# B&R Automation Studio project Projekt_BuR
Automation Studio 4.11.2.75; technology packages: exosTechnology 2.1.0, mapp 5.18.0, mappCockpit 5.18.0, mappControl 5.18.0, mappView 5.18.1

## Configuration X20CP3586

CPU X20CP3586, AutomationRuntime C4.92, Build 4.1.2, Safety 0.0, Vc V4.72.5

### Task classes (Cpu.sw)
```
Cyclic#1 (cycle 2000 us, tolerance 0 us):
  TempContro <- Control.TempControl.prg
  TempScalin <- TempScaling.prg
Cyclic#3:
  MQTT <- Control.MQTT.prg
Cyclic#4:
  Alarm <- Control.Alarm.prg
  Recipe <- Control.Recipe.prg
  OEE <- Control.OEE.prg
  AuditTrail <- Control.AuditTrail.prg
  MpReport1 <- Control.MpReport.prg
  DataMgmt <- Control.DataMgmt.prg
  VisuAdj <- Control.VisuAdj.prg
  FileCtrl <- Control.FileCtrl.prg
Binaries: udbdef, FWRules, TCData, TCLang, arsvcreg, mvLoader, mCoWebSc, arflatprv, arcoal, iomap, ashwac, Role, sysconf, arconfig, asfw, User, ashwd, HeatZone3, HeatZone2, HeatZone1, HeatZone4, TC, HeatGroup, ConfigAudi, ConfigAHis, ConfigAlar, ConfigData, ConfigOEE, report, ConfigFile, RecipeCon, Config
Libraries: CoTrace, AsZip, FileIO, runtime, MpAlarmX, MpBase, astime, MpServer, MpTemp, IotMqtt, AsIecCon, ArCert, sys_lib, AsHW, AsETH, ArEventLog, AsIODiag, AsBrStr, standard, MpAudit, MpReport, AsMath, MpOee, MpData, DataObj, brsystem, MpFile, MpRecipe, MTBasics, MTTypes, arssl, aruser, asusb, MpUserX
```

### Hardware
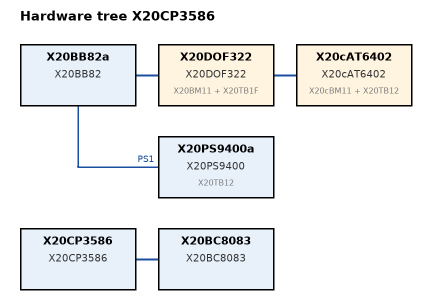
```
X20BB82a : X20BB82 v1.1.0.0
X20BC8083 : X20BC8083 v2.12.0.0  [PLK1 -> X20CP3586.IF3 (NodeNumber=1) [Cable Type=PowerlinkCable, Length=10, Version=1.0.0.3]; SL -> X20BB82a.SL1]
  Supervision = off
X20BM11a : X20BM11 v1.1.0.0  [X2X1 -> X20BB82a.IF1]
X20CP3586 : X20CP3586 v1.10.0.0
  Connector IF2:
    ActivateDevice = 1
    Mode = Manual
    InternetAddress = 192.168.0.22
    SubnetMask = 255.255.255.0
    ActivateSnmp = 2
  Connector IF3:
    CycleTime = 400
  ConfigurationID = Projekt_BuR_X20CP3586
  TimerDeviceType = EPLX2X
  TimerDevice = X20CP3586.IF3
  TaskClassIdleTime = 2000
  Cyclic1Duration = 2000
  Cyclic1Tolerance = 0
  FileDevice1
  FileDeviceName1 = AUDIT
  FileDevicePath1 = F:/BRAudit
  FileDevice2
  FileDeviceName2 = DATA
  FileDevicePath2 = F:/BRmappData
  FileDevice3
  FileDeviceName3 = PDF
  FileDevicePath3 = F:/PDF
  FileDevice4
  FileDeviceName4 = DISK
  FileDevicePath4 = F:/
  FileDevice5
  FileDeviceName5 = RECIPE
  FileDevicePath5 = F:/BrRecipe
  FileDevice6
  FileDeviceName6 = BRVisu
  FileDevicePath6 = C:/ADDONS/DATA/IAT_Data/wwwRoot/BRVisu
  TimeZone = 160
  ActivateDaylightSavingTime = 1
  FtpUser1
  FtpUsername1 = Admin
  FtpUserPassword1 = 5wGvT8auoKyFZyijp5IHEBz1PpSmCNNWGV/kzWv0+cU=
  FtpUserSalt1 = OGipJzaF
  FTPAccessRight1 = 0
  FTPdevice1 = ALL
  ActivateOpcUa = 1
  OpcUaInformationModels_PV_Version = 1
X20DOF322 : X20DOF322 v1.5.0.0  [SS1 -> X20TB1F1.SS; SL -> X20BM11a.SL1]
  Supervision = off
X20PS9400a : X20PS9400 v1.7.0.0  [SS1 -> X20TB12.SS; PS -> X20BB82a.PS1]
  Supervision = off
X20TB12 : X20TB12 v1.0.0.0
X20TB12a : X20TB12 v1.0.0.0
X20TB1F1 : X20TB1F v1.0.0.0
X20cAT6402 : X20cAT6402 v1.2.0.0  [SS1 -> X20TB12a.SS; SL -> X20cBM11a.SL1]
  Supervision = off
  DisableChannel01 = on
  DisableChannel02 = on
X20cBM11a : X20cBM11 v1.1.0.0  [X2X1 -> X20BM11a.X2X2]
```

### ConfigAlar.mpalarmxcore - X20CP3586/mappServices/ConfigAlar.mpalarmxcore
```
Element gAlarmXCore (Type=mpalarmxcore)
  mapp.AlarmX.Core:
    Mapping:
      [0]:
        Alarm = High Temperature1#HighHigh
        [0] = Reaction
          Name = StatusIdle
      [1]:
        Alarm = High Temperature2#HighHigh
        [0] = Reaction
          Name = StatusIdle
      [2]:
        Alarm = High Temperature3#HighHigh
        [0] = Reaction
          Name = StatusIdle
      [3]:
        Alarm = High Temperature4#HighHigh
        [0] = Reaction
          Name = StatusIdle
      [4]:
        Alarm = X20BC8083
        [0] = Reaction
          Name = StatusIdle
      [5]:
        Alarm = X20PS9400a
        [0] = Reaction
          Name = StatusIdle
      [6]:
        Alarm = X20DOF322
        [0] = Reaction
          Name = StatusIdle
      [7]:
        Alarm = X20cAT6402
        [0] = Reaction
          Name = StatusIdle
      [8]:
        Alarm =  Fan failure1
        [0] = Reaction
          Name = StatusIdle
      [9]:
        Alarm =  Fan failure2
        [0] = Reaction
          Name = StatusIdle
      [10]:
        Alarm =  Fan failure3
        [0] = Reaction
          Name = StatusIdle
      [11]:
        Alarm =  Fan failure4
        [0] = Reaction
          Name = StatusIdle
      [12]:
        Alarm = Sensor failure1
        [0] = Reaction
          Name = StatusIdle
      [13]:
        Alarm = Sensor failure2
        [0] = Reaction
          Name = StatusIdle
      [14]:
        Alarm = Sensor failure3
        [0] = Reaction
          Name = StatusIdle
      [15]:
        Alarm = Sensor failure4
        [0] = Reaction
          Name = StatusIdle
  mapp.AlarmX.Core.Configuration:
    [0]:
      Name = High Temperature1
      Message = {$IAT/Alarms/HT1Message}
      Code = 1037
      Behavior = LevelMonitoring
        Monitoring:
          MonitoredPV = ::gTemp1
          HighLimitEnable = Dynamic
            LimitPV = ::Alarms.TempAlarmLimit
            HighHighLimitEnable = Dynamic
              LimitPV = ::Alarms.TempMaxAlarmLimit
              LimitText = HighHigh
    [1]:
      Name = High Temperature2
      Message = {$IAT/Alarms/HT2Message}
      Code = 1038
      Behavior = LevelMonitoring
        Monitoring:
          MonitoredPV = ::gTemp2
          HighLimitEnable = Dynamic
            LimitPV = ::Alarms.TempAlarmLimit
            HighHighLimitEnable = Dynamic
              LimitPV = ::Alarms.TempMaxAlarmLimit
              LimitText = HighHigh
    [2]:
      Name = High Temperature3
      Message = {$IAT/Alarms/HT3Message}
      Code = 1039
      Behavior = LevelMonitoring
        Monitoring:
          MonitoredPV = ::gTemp3
          HighLimitEnable = Dynamic
            LimitPV = ::Alarms.TempAlarmLimit
            HighHighLimitEnable = Dynamic
              LimitPV = ::Alarms.TempMaxAlarmLimit
              LimitText = HighHigh
    [3]:
      Name = High Temperature4
      Message = {$IAT/Alarms/HT4Message}
      Code = 1040
      Behavior = LevelMonitoring
        Monitoring:
          MonitoredPV = ::gTemp4
          HighLimitEnable = Dynamic
            LimitPV = ::Alarms.TempAlarmLimit
            HighHighLimitEnable = Dynamic
              LimitPV = ::Alarms.TempMaxAlarmLimit
              LimitText = HighHigh
    [4]:
      Name = X20BC8083
      Message = {$IAT/Alarms/X20BC8083}
      Code = 1308
      Behavior = DiscreteValueMonitoring
        Monitoring:
          MonitoredPV = ::Alarms.first_module
          TriggerValues:
            [0] = 0
    [5]:
      Name = X20PS9400a
      Message = {$IAT/Alarms/X20PS9400a}
      Code = 1309
      Behavior = DiscreteValueMonitoring
        Monitoring:
          MonitoredPV = ::Alarms.second_module
          TriggerValues:
            [0] = 0
    [6]:
      Name = X20DOF322
      Message = {$IAT/Alarms/X20DOF322}
      Code = 1310
      Behavior = DiscreteValueMonitoring
        Monitoring:
          MonitoredPV = ::Alarms.third_module
          TriggerValues:
            [0] = 0
    [7]:
      Name = X20cAT6402
      Message = {$IAT/Alarms/X20cAT6402}
      Code = 1311
      Behavior = DiscreteValueMonitoring
        Monitoring:
          MonitoredPV = ::Alarms.fourth_module
          TriggerValues:
            [0] = 0
    [8]:
      Name =  Fan failure1
      Message = {$IAT/Alarms/FanAlarmMessage1}
      Code = 1446
      Behavior = DiscreteValueMonitoring
        Monitoring:
          MonitoredPV = ::Alarms.FanAlarm1
          TriggerValues:
            [0] = 1
    [9]:
      Name =  Fan failure2
      Message = {$IAT/Alarms/FanAlarmMessage2}
      Code = 1447
      Behavior = DiscreteValueMonitoring
        Monitoring:
          MonitoredPV = ::Alarms.FanAlarm2
          TriggerValues:
            [0] = 1
    [10]:
      Name =  Fan failure3
      Message = {$IAT/Alarms/FanAlarmMessage3}
      Code = 1448
      Behavior = DiscreteValueMonitoring
        Monitoring:
          MonitoredPV = ::Alarms.FanAlarm3
          TriggerValues:
            [0] = 1
    [11]:
      Name =  Fan failure4
      Message = {$IAT/Alarms/FanAlarmMessage4}
      Code = 1449
      Behavior = DiscreteValueMonitoring
        Monitoring:
          MonitoredPV = ::Alarms.FanAlarm4
          TriggerValues:
            [0] = 1
    [12]:
      Name = Sensor failure1
      Message = {$IAT/Alarms/HeaterAlarmMess1}
      Severity = 1455
      Behavior = DiscreteValueMonitoring
        Monitoring:
          MonitoredPV = ::Alarms.HeaterAlarm1
          TriggerValues:
            [0] = 1
    [13]:
      Name = Sensor failure2
      Message = {$IAT/Alarms/HeaterAlarmMess2}
      Severity = 1456
      Behavior = DiscreteValueMonitoring
        Monitoring:
          MonitoredPV = ::Alarms.HeaterAlarm2
          TriggerValues:
            [0] = 1
    [14]:
      Name = Sensor failure3
      Message = {$IAT/Alarms/HeaterAlarmMess3}
      Severity = 1457
      Behavior = DiscreteValueMonitoring
        Monitoring:
          MonitoredPV = ::Alarms.HeaterAlarm3
          TriggerValues:
            [0] = 1
    [15]:
      Name = Sensor failure4
      Message = {$IAT/Alarms/HeaterAlarmMess4}
      Severity = 1458
      Behavior = DiscreteValueMonitoring
        Monitoring:
          MonitoredPV = ::Alarms.HeaterAlarm4
          TriggerValues:
            [0] = 1
```

### ConfigUser.mpuserx - X20CP3586/mappServices/ConfigUser.mpuserx
```
Element UserMgmtX (Type=mpuserx)
  ServerSettings:
    Server:
      AdditionalUserData:
        [0] = mail
        [1] = telephoneNumber
  Users:
    DefUser#1:
      id = Administrator
    DefUser#2:
      id = Operator
    DefUser#3:
      id = a
    DefUser#4:
      id = Anonymous
  Groups:
    DefGroup#1:
      id = Administrators
      level = 100
      admin = TRUE
      rights:
        [0] = FullAccess
    DefGroup#2:
      id = Operators
      level = 30
    DefGroup#3:
      id = Everyone
      level = 3
```

## Logical view

Binary libraries used (declarations not repeated): operator, runtime, astime, AsIecCon, CoTrace, AsZip, FileIO, MpAlarmX, MpBase, MpServer, MpTemp, IotMqtt, ArCert, sys_lib, AsHW, AsETH, ArEventLog, AsIODiag, AsBrStr, standard, MpOee, MpAudit, MpReport, AsMath, MpData, DataObj, brsystem, MpFile, MpRecipe, MTBasics, MTTypes, MpUserX, ExOS, ExDeploy, ExData, AsIoTime

### ControlTypes.typ
```iecst
TYPE
	AUTOMATIC_MODE_STATE :
		( (*Step of automatic mode*)
		STEP_INIT,
		STEP1,
		STEP2,
		STEP3,
		STEP4,
		STEP5
		);
	ZONE_WORKING_STATE :
		( (*Working state of each zone*)
		STATE_IDLE_ZONE,
		STATE_HEATING,
		STATE_COOLING
		);
	MACHINE_WORKING_STATE :
		( (*Working state of whole machine*)
		STATE_IDLE,
		STATE_TUNING,
		STATE_WORKING_MANUAL,
		STATE_WORKING_AUTOMATIC,
		STATE_ERROR,
		STATE_STOP
		);
	MACHINE_PARAMETERS : 	STRUCT  (*Machine parameters - structed*)
		Temp1 : REAL;
		Temp2 : REAL;
		Temp3 : REAL;
		Temp4 : REAL;
		Time1 : TIME;
		Time2 : TIME;
		Time3 : TIME;
		Time4 : TIME;
		Time5 : TIME;
	END_STRUCT;
	Alarm_struct : 	STRUCT
		Pending : UDINT := 0;
		Active : UDINT := 0;
		FanAlarm4 : BOOL;
		FanAlarm3 : BOOL;
		FanAlarm2 : BOOL;
		FanAlarm1 : BOOL;
		HeaterAlarm4 : BOOL;
		HeaterAlarm3 : BOOL;
		HeaterAlarm2 : BOOL;
		HeaterAlarm1 : BOOL;
		fourth_module : BOOL;
		third_module : BOOL;
		second_module : BOOL;
		first_module : BOOL;
		TempMaxAlarmLimit : REAL := 50;
		TempAlarmLimit : REAL := 40;
		ActiveAlarms : STRING[512] := 'test';
	END_STRUCT;
	OEE_Struct : 	STRUCT
		IdealCycleTime : STRING[80];
		OEE : REAL;
		Quality : REAL;
		Performance : REAL;
		Availability : REAL;
		RejectCounter : UDINT;
		PieceCounter : UDINT;
	END_STRUCT;
END_TYPE
```

### ControlVariables.var
```iecst
(*Temperature setpoints to all zones.*)
VAR
	SetTemp1 : REAL := 30; (*Set temperature for zone 1.*)
	SetTemp2 : REAL := 30; (*Set temperature for zone 2.*)
	SetTemp3 : REAL := 30; (*Set temperature for zone 3.*)
	SetTemp4 : REAL := 30; (*Set temperature for zone 4.*)
END_VAR
(*Temperature tuning setpoints to all zones.*)
VAR
	SetTempHeatTuning1 : REAL := 100; (*Set heating temperature for zone 1.*)
	SetTempHeatTuning2 : REAL := 100; (*Set heating temperature for zone 2.*)
	SetTempHeatTuning3 : REAL := 100; (*Set heating temperature for zone 3.*)
	SetTempHeatTuning4 : REAL := 100; (*Set  heating temperature for zone 4.*)
	SetTempCoolTuning1 : REAL := 30; (*Set cooling temperature for zone 1.*)
	SetTempCoolTuning2 : REAL := 30; (*Set cooling temperature for zone 2.*)
	SetTempCoolTuning3 : REAL := 30; (*Set cooling temperature for zone 3.*)
	SetTempCoolTuning4 : REAL := 30; (*Set cooling temperature for zone 4.*)
END_VAR
(*Machine status - step.*)
VAR
	STATUS : MACHINE_WORKING_STATE := STATE_IDLE; (*Whole machine working status.*)
END_VAR
(*Zones status*)
VAR
	ZoneStatus : ARRAY[0..ELEMENTS_NUMBER] OF ZONE_WORKING_STATE; (*Each zone working status.*)
END_VAR
(*Temperature controller functionblocks.*)
VAR
	TempControllerPar : ARRAY[0..ELEMENTS_NUMBER] OF MpTempControllerParType; (*Array of 4 additions to controllers*)
	TempController : ARRAY[0..ELEMENTS_NUMBER] OF MpTempController; (*Array of 4 controllers - one for each zone*)
	TempGroup : MpTempGroup; (*Controller group*)
	TempGroupPar : MpTempGroupParType; (*Adition to controllergroup*)
END_VAR
(*Const elements.*)
VAR CONSTANT
	ELEMENTS_NUMBER : USINT := 3; (*Numbers of controling zones - 4 (0,1,2,3)*)
END_VAR
(*Machine working type*)
VAR
	Automatic_work : BOOL := FALSE; (*Enable automatic work mode.*)
	Manual_work : BOOL := FALSE; (*Enable manual work mode.*)
	TuneEnable : BOOL := FALSE; (*Enable tune work mode.*)
END_VAR
(*Manual control*)
VAR
	EnableZone1 : BOOL := TRUE; (*Enable zone 1.*)
	EnableZone2 : BOOL := TRUE; (*Enable zone 2.*)
	EnableZone3 : BOOL := TRUE; (*EnableZone 3.*)
	EnableZone4 : BOOL := TRUE; (*Enable zone 4.*)
END_VAR
(*Automatic control*)
VAR
	AutoStep : AUTOMATIC_MODE_STATE := STEP_INIT;
	TimeStep1 : TIME := T#5s; (*Min time of step 1*)
	TimeStep2 : TIME := T#5s; (*Min time of step 2*)
	TimeStep3 : TIME := T#5s; (*Min time of step 3*)
	TimeStep4 : TIME := T#5s; (*Min time of step 4*)
	TimeStep5 : TIME := T#5s; (*Min time of step 5*)
	TimStep1 : TON; (*Timer for step 1 in automatic work.*)
	TimStep2 : TON; (*Timer for step 2 in automatic work.*)
	TimStep3 : TON; (*Timer for step 3 in automatic work.*)
	TimStep4 : TON; (*Timer for step 4 in automatic work.*)
	TimStep5 : TON; (*Timer in step 5 for automatic work.*)
	CycleNumber : DINT := 0; (*Number of full done cycles in automatic work.*)
END_VAR
(*Simulation mode*)
VAR
	SimulateZone1Enable : BOOL := FALSE; (*Simulation enable of zone 1.*)
	SimulateZone2Enable : BOOL := FALSE; (*Simulation enable of zone 2.*)
	SimulateZone3Enable : BOOL := FALSE; (*Simulation enable of zone 3.*)
	SimulateZone4Enable : BOOL := FALSE; (*Simulation enable of zone 4.*)
END_VAR
(*Tuning parameters HEAT*)
VAR RETAIN
	PIDProportionaGainHEAT : ARRAY[0..ELEMENTS_NUMBER] OF REAL := [49.3,45.56,31.29,35.25];
	PIDIntegrationTimeHEAT : ARRAY[0..ELEMENTS_NUMBER] OF REAL := [64.92,75.59,95.21,101.41];
	PIDFilterTimeHEAT : ARRAY[0..ELEMENTS_NUMBER] OF REAL := [0.682,0.762,0.99,1.06];
	PIDDerivativeTimeHEAT : ARRAY[0..ELEMENTS_NUMBER] OF REAL := [6.82,7.62,9.99,10.64];
END_VAR
(*Tuning parameters COOL*)
VAR RETAIN
	PIDProportionaGainCOOL : ARRAY[0..ELEMENTS_NUMBER] OF REAL := [20.96,27.64,18.07,26.18];
	PIDIntegrationTimeCOOL : ARRAY[0..ELEMENTS_NUMBER] OF REAL := [68.71,46.86,80.30,51.64];
	PIDDerivativeTimeCOOL : ARRAY[0..ELEMENTS_NUMBER] OF REAL := [7.22,4.92,8.43,5.42];
	PIDFilterTimeCOOL : ARRAY[0..ELEMENTS_NUMBER] OF REAL := [0.72,0.49,0.84,0.54];
END_VAR
(*Alarm*)
VAR
	Alarms : Alarm_struct;
	MpAlarmXCore_0 : MpAlarmXCore;
END_VAR
(*OEE*)
VAR
	OEE : OEE_Struct;
END_VAR
(* ########## MQTT communication variables ########### *)
(*PWM % Heater Zone 1  ->  TempController[0].HeatValue*)
(*PWM % Heater Zone 2  ->  TempController[1].HeatValue*)
(*PWM % Heater Zone 3  ->  TempController[2].HeatValue*)
(*PWM % Heater Zone 4  ->  TempController[3].HeatValue*)
(*PWM % FAN Zone 1  ->  TempController[0].CoolValue*)
(*PWM % FAN Zone 2  ->  TempController[1].CoolValue*)
(*PWM % FAN Zone 3  ->  TempController[2].CoolValue*)
(*PWM % FAN Zone 4  ->  TempController[3].CoolValue*)
(*Set Temperature Zone 1  ->  SetTemp1*)
(*Set Temperature Zone 2  ->  SetTemp2*)
(*Set Temperature Zone 3  ->  SetTemp3*)
(*Set Temperature Zone 4  ->  SetTemp4*)
(*Actual Temperature Zone 1  ->  gTemp1*)
(*Actual Temperature Zone 2  ->  gTemp2*)
(*Actual Temperature Zone 3  ->  gTemp3*)
(*Actual Temperature Zone 4  ->  gTemp4*)
(*Status dzialania calej maszyny -> STATUS (typ: MACHINE_WORKING_STATE)*)
(*Status dzialania trybu automatycznego -> AutoStep (typ: AUTOMATIC_MODE_STATUS)*)
(*Status dzialania strefy 1 -> ZoneStatus[0] (typ: ZONE_WORKING_STATUS)*)
(*Status dzialania strefy 2 -> ZoneStatus[1] (typ: ZONE_WORKING_STATUS)*)
(*Status dzialania strefy 3 -> ZoneStatus[2] (typ: ZONE_WORKING_STATUS)*)
(*Status dzialania strefy 4 -> ZoneStatus[3] (typ: ZONE_WORKING_STATUS)*)
(*Ilosc wykonanych cykli w trybie automatycznym -> CycleNumber*)
(*//////////////////////////////Machine parameters*)
VAR
	ParametersMachine : MACHINE_PARAMETERS;
END_VAR
(*Recipe*)
VAR
	RecipeListName : ARRAY[0..9] OF STRING[255];
END_VAR
(*Audit*)
VAR
	MpAuditTrail_0 : MpAuditTrail;
	MessageVar : WSTRING[100] := "Hello World";
END_VAR
(*pid pwm*)
VAR
	MTBasicsPID_HEAT : ARRAY[0..ELEMENTS_NUMBER] OF MTBasicsPID;
	ParameterTypePIDHEAT : ARRAY[0..ELEMENTS_NUMBER] OF MTPIDParametersType;
	MTBasicsPID_COLD : ARRAY[0..ELEMENTS_NUMBER] OF MTBasicsPID;
	ParameterTypePIDCOLD : ARRAY[0..ELEMENTS_NUMBER] OF MTPIDParametersType;
	MTBasicsPWM_HEAT : ARRAY[0..ELEMENTS_NUMBER] OF MTBasicsPWM;
	MTBasicsPWM_COLD : ARRAY[0..ELEMENTS_NUMBER] OF MTBasicsPWM;
	Temp1Alarm : REAL;
	Temp2Alarm : REAL;
END_VAR
(**)
```

### Program Logical/Control/Alarm

#### Main.st
```iecst
PROGRAM _INIT
	(* Insert code here *)
	MpAlarmXCore_0.MpLink :=  ADR(gAlarmXCore);
	MpAlarmXCore_0.Enable := TRUE;
	MpAlarmXHistory_0.MpLink :=  ADR(gAlarmXHistory);
	MpAlarmXHistory_0.Enable := TRUE;
	MpAlarmXCore_0();
	MpAlarmXHistory_0();
	mpAlarmXlist.MpLink :=ADR(gAlarmXCore);
	mpAlarmXlist.Enable := TRUE;
	mpAlarmXlist.UIConnect := ADR(mpAlarmXlistConnect);
	mpAlarmXlist.UISetup := MpAlarmXlistSetup;
	//initialization
	Temp1Alarm;
	Temp2Alarm;
END_PROGRAM

PROGRAM _CYCLIC
	(* Insert code here *)
	MpAlarmXCore_0();
	MpAlarmXHistory_0();
	mpAlarmXlist();
	IF MpAlarmXCheckReaction(gAlarmXCore,'StatusIdle') THEN
		Automatic_work := FALSE;
		Manual_work := FALSE;
		TuneEnable := FALSE;
		gStart := FALSE;
		gSTOP := FALSE;
		gError := FALSE;
		STATUS := STATE_IDLE;
	END_IF;

	Alarms.Pending := MpAlarmXCore_0.PendingAlarms;
	Alarms.Active :=  MpAlarmXCore_0.ActiveAlarms;
	Alarms.ActiveAlarms := '';
	FOR i:=0 TO 49 BY 1 DO
		IF NOT (mpAlarmXlistConnect.AlarmList.Code[i]=0) THEN
			stringBuffer := UDINT_TO_STRING(mpAlarmXlistConnect.AlarmList.Code[i]);
			brsstrcat(ADR(Alarms.ActiveAlarms),ADR(stringBuffer));

			stringBuffer := ';';
			brsstrcat(ADR(Alarms.ActiveAlarms),ADR(stringBuffer));

			stringBuffer := WSTRING_TO_STRING(mpAlarmXlistConnect.AlarmList.Message[i]);
			brsstrcat(ADR(Alarms.ActiveAlarms),ADR(stringBuffer));

			stringBuffer := ';';
			brsstrcat(ADR(Alarms.ActiveAlarms),ADR(stringBuffer));

			stringBuffer := (mpAlarmXlistConnect.AlarmList.Timestamp[i]);
			brsstrcat(ADR(Alarms.ActiveAlarms),ADR(stringBuffer));

			stringBuffer := ';';
			brsstrcat(ADR(Alarms.ActiveAlarms),ADR(stringBuffer));

			stringBuffer := BOOL_TO_STRING(mpAlarmXlistConnect.AlarmList.StateAcknowledged[i]);
			brsstrcat(ADR(Alarms.ActiveAlarms),ADR(stringBuffer));

			stringBuffer := ';';
			brsstrcat(ADR(Alarms.ActiveAlarms),ADR(stringBuffer));

			stringBuffer := BOOL_TO_STRING(mpAlarmXlistConnect.AlarmList.StateActive[i]);
			brsstrcat(ADR(Alarms.ActiveAlarms),ADR(stringBuffer));

			IF NOT (i=49 OR mpAlarmXlistConnect.AlarmList.Code[i+1]=0) THEN
				stringBuffer :=',';
				brsstrcat(ADR(Alarms.ActiveAlarms),ADR(stringBuffer));
			END_IF
		END_IF
	END_FOR
END_PROGRAM

PROGRAM _EXIT
	(* Insert code here *)
	MpAlarmXCore_0.Enable := FALSE;
	MpAlarmXHistory_0.Enable := FALSE;
	mpAlarmXlist.Enable := FALSE;
	mpAlarmXlist();
	MpAlarmXCore_0();
	MpAlarmXHistory_0();
END_PROGRAM
```

### Program Logical/Control/MQTT

#### Init.st
```iecst
ACTION Init:
	IotMqttParameters.ServerUri				:= '10.48.10.127';
	IotMqttParameters.Port					:= 1883;
	IotMqttParameters.ClientID				:= 'PLC';

	IotMqttClient_0.Enable					:= TRUE;
	IotMqttClient_0.Connect					:= TRUE;
	IotMqttClient_0.IotMqttLink 			:= ADR(IotMqttLink);
	IotMqttClient_0.Parameters				:= IotMqttParameters;

	IotMqttPublish_0.Enable					:= TRUE;
	IotMqttPublish_0.IotMqttLink			:= ADR(IotMqttLink);

	TopicCounter.PV := NR_OF_TOPICS-1;
END_ACTION
```

#### Main.st
```iecst
PROGRAM _INIT
	(* Insert code here *)
	Init;
END_PROGRAM

PROGRAM _CYCLIC
	(* Insert code here	*)
	UpdateStructs;
	doSend := NOT doSend;
	IotMqttPublish_0.Send :=FALSE;
	TopicCounter.CU := FALSE;

	TopicSelectionTransmision;

	TopicCounter();
	IotMqttClient_0();
	IotMqttPublish_0();
END_PROGRAM

PROGRAM _EXIT
	(* Insert code here *)
	IotMqttClient_0(Enable := FALSE);
	IotMqttPublish_0(Enable := FALSE);
	IotMqttClient_0();
	IotMqttPublish_0();
END_PROGRAM
```

#### UpdateStructs.st
```iecst
ACTION UpdateStructs:
	IF SimulateZone1Enable THEN
		Fans.Fan1 := TempController[0].Info.Simulation.CoolValue;
		Heaters.Heater1 := TempController[0].Info.Simulation.HeatValue;
		Temps.Temp1 := TempController[0].Info.Simulation.ActualTemperature;
	ELSE
		Fans.Fan1 := TempController[0].CoolValue;
		Heaters.Heater1 := TempController[0].HeatValue;
		Temps.Temp1 := gTemp1;
	END_IF;

	IF SimulateZone2Enable THEN
		Fans.Fan2 := TempController[1].Info.Simulation.CoolValue;
		Heaters.Heater2 := TempController[1].Info.Simulation.HeatValue;
		Temps.Temp2 := TempController[1].Info.Simulation.ActualTemperature;
	ELSE
		Fans.Fan2 := TempController[1].CoolValue;
		Heaters.Heater2 := TempController[1].HeatValue;
		Temps.Temp2 := gTemp2;
	END_IF;

	IF SimulateZone3Enable THEN
		Fans.Fan3 := TempController[2].Info.Simulation.CoolValue;
		Heaters.Heater3 := TempController[2].Info.Simulation.HeatValue;
		Temps.Temp3 := TempController[2].Info.Simulation.ActualTemperature;
	ELSE
		Fans.Fan3 := TempController[2].CoolValue;
		Heaters.Heater3 := TempController[2].HeatValue;
		Temps.Temp3 := gTemp3;
	END_IF;

	IF SimulateZone4Enable THEN
		Fans.Fan4 := TempController[3].Info.Simulation.CoolValue;
		Heaters.Heater4 := TempController[3].Info.Simulation.HeatValue;
		Temps.Temp4 := TempController[3].Info.Simulation.ActualTemperature;
	ELSE
		Fans.Fan4 := TempController[3].CoolValue;
		Heaters.Heater4 := TempController[3].HeatValue;
		Temps.Temp4 := gTemp4;
	END_IF;

//	Fans.Fan1 := TempController[0].Info.Simulation.CoolValue;
//	Fans.Fan2 := TempController[1].CoolValue;
//	Fans.Fan3 := TempController[2].CoolValue;
//	Fans.Fan4 := TempController[3].CoolValue;
//
//	Temps.Temp1 := TempController[0].Info.Simulation.ActualTemperature;
//	Temps.Temp2 := gTemp2;
//	Temps.Temp3 := gTemp3;
//	Temps.Temp4 := gTemp4;

	SetPoint.SetPoint1 := SetTemp1;
	SetPoint.SetPoint2 := SetTemp2;
	SetPoint.SetPoint3 := SetTemp3;
	SetPoint.SetPoint4 := SetTemp4;

	Zones.Zone1 := ZoneStatus[0];
	Zones.Zone2 := ZoneStatus[1];
	Zones.Zone3 := ZoneStatus[2];
	Zones.Zone4 := ZoneStatus[3];

//	Heaters.Heater1 := TempController[0].Info.Simulation.HeatValue;
//	Heaters.Heater2 := TempController[1].HeatValue;
//	Heaters.Heater3 := TempController[2].HeatValue;
//	Heaters.Heater4 := TempController[3].HeatValue;

	MachineState.Machine_state := STATUS;
END_ACTION
```
